// TIA Portal project "TruongKhuongDuy_20151451_DoanPLC_V17" (V17)
// Vorlageprojekt für das Buch mit Zielsystem S7-1200

(* hardware
DEVICE "S7-1200-Station_1"  S7-1200 Station
   slot 0: "Baugruppenträger_0"  Rack  V1.0
   slot 1: "PLC_1"  CPU 1211C DC/DC/DC  6ES7 211-1AE40-0XB0  V4.1
*)

// ===== PLC "PLC_1"  CPU 1211C DC/DC/DC =====

VAR_GLOBAL   // PLC tag table "Standard-Variablentabelle"
   "At exit" AT %I0.0 : Bool;
   "Start" AT %I0.1 : Bool;
   "Reset" AT %I0.2 : Bool;
   "Stop" AT %I0.3 : Bool;
   "Auto" AT %M20.0 : Bool;
   "Sensor 1" AT %I0.6 : Bool;
   "Sensor 4" AT %I0.7 : Bool;
   "Sensor 2" AT %I1.0 : Bool;
   "Sensor 3" AT %I1.1 : Bool;
   "Sensor box" AT %I1.2 : Bool;
   "Clamped" AT %I1.3 : Bool;
   "Limit" AT %I1.4 : Bool;
   "Detected 1" AT %I1.5 : Bool;
   "Moving Z1" AT %I1.6 : Bool;
   "Moving X1" AT %I1.7 : Bool;
   "Clamped 2" AT %I2.0 : Bool;
   "Limit 2" AT %I2.1 : Bool;
   "Detected 2" AT %I2.2 : Bool;
   "Moving Z2" AT %I2.3 : Bool;
   "Moving X2" AT %I2.4 : Bool;
   "Out Vision sensor" AT %ID30 : DInt;
   "Entry Converyor" AT %Q0.0 : Bool;
   "Alam siren" AT %Q0.1 : Bool;
   "Exit converyor" AT %Q0.2 : Bool;
   "Sotter 1 turn" AT %Q0.3 : Bool;
   "Sotter 1 belt" AT %Q0.4 : Bool;
   "Sotter 2 turn" AT %Q0.5 : Bool;
   "Sotter 2 belt" AT %Q0.6 : Bool;
   "Sotter 3 turn" AT %Q0.7 : Bool;
   "Sotter 3 belt" AT %Q1.0 : Bool;
   "Start light" AT %Q1.1 : Bool;
   "Reset light" AT %Q1.2 : Bool;
   "Stop light" AT %Q1.3 : Bool;
   "Belt Conveyor 1" AT %Q1.4 : Bool;
   "Belt Conveyor 2" AT %Q1.5 : Bool;
   "Box Conveyor" AT %Q1.6 : Bool;
   "Clamp 1" AT %Q1.7 : Bool;
   "Raise 1" AT %Q2.0 : Bool;
   "Mover Z1" AT %Q2.1 : Bool;
   "Mover X1" AT %Q2.2 : Bool;
   "Grab 1" AT %Q2.3 : Bool;
   "Clamp 2" AT %Q2.4 : Bool;
   "Raise 2" AT %Q2.5 : Bool;
   "Mover Z2" AT %Q2.6 : Bool;
   "Mover X2" AT %Q2.7 : Bool;
   "Grab 2" AT %Q3.0 : Bool;
   "Start Light ( Green)" AT %Q3.1 : Bool;
   "Reset Light ( Yellow)" AT %Q3.2 : Bool;
   "Stop Light ( Red)" AT %Q3.3 : Bool;
   "Stop Blade 1" AT %Q3.4 : Bool;
   "Counter 1" AT %QD30 : DInt;
   "Counter 2" AT %QD34 : DInt;
   "Counter 3" AT %QD38 : DInt;
   "Counter 4" AT %QD42 : DInt;
   "TG1" AT %M0.0 : Bool;
   "TG4" AT %M0.1 : Bool;
   "TG3" AT %M1.1 : Bool;
   "TG STOP CG" AT %M0.2 : Bool;
   "TG5" AT %M0.5 : Bool;
   "TG6" AT %M0.3 : Bool;
   "Tag_3" AT %M100.0 : Bool;
   "Tag_1" AT %M100.1 : Bool;
   "CB sensor4" AT %M100.3 : Bool;
   "Tag_2" AT %M101.1 : Bool;
   "Tag_4" AT %M100.2 : Bool;
   "Tag_5" AT %M100.4 : Bool;
   "Tag_6" AT %M100.7 : Bool;
   "Tag_8" AT %M100.6 : Bool;
   "Tag_9" AT %M200.0 : Bool;
   "Tag_10" AT %M200.1 : Bool;
   "Tag_11" AT %M200.2 : Bool;
   "Tag_12" AT %M200.3 : Bool;
   "Tag_13" AT %M200.4 : Bool;
   "Tag_14" AT %M200.7 : Bool;
   "Tag_15" AT %M200.6 : Bool;
   "Tag_16" AT %QD46 : DWord;
   "Tag_17" AT %M100.5 : Bool;
   "M_Stop" AT %M150.1 : Bool;
   "M_Reset" AT %M150.2 : Bool;
   "M_Start" AT %M150.0 : Bool;
   "M_exit" AT %M150.3 : Bool;
   "M_sensor1" AT %M150.4 : Bool;
   "M_sensor2" AT %M150.5 : Bool;
   "M_sensor3" AT %M150.6 : Bool;
   "M_sensor4" AT %M150.7 : Bool;
   "M_sensorbox" AT %M151.0 : Bool;
   "M_Auto" AT %M151.1 : Bool;
   "Tag_18" AT %M151.2 : Bool;
   "Tag_7" AT %M210.0 : Bool;
   "Emergency stop" AT %I0.4 : Bool;
END_VAR

// folder: System blocks/Program resources

DATA_BLOCK "IEC_Timer_0_DB"   // DB1
{ S7_Optimized_Access := 'TRUE' }
AUTHOR : Simatic
FAMILY : IEC
NAME : IEC_TMR
VERSION : 1.0
// stored: InstanceOfName IEC_TIMER
"IEC_TIMER"
BEGIN
END_DATA_BLOCK

DATA_BLOCK "IEC_Timer_0_DB_1"   // DB2
{ S7_Optimized_Access := 'TRUE' }
AUTHOR : Simatic
FAMILY : IEC
NAME : IEC_TMR
VERSION : 1.0
// stored: InstanceOfName IEC_TIMER
"IEC_TIMER"
BEGIN
END_DATA_BLOCK

DATA_BLOCK "IEC_Timer_0_DB_2"   // DB3
{ S7_Optimized_Access := 'TRUE' }
AUTHOR : Simatic
FAMILY : IEC
NAME : IEC_TMR
VERSION : 1.0
// stored: InstanceOfName IEC_TIMER
"IEC_TIMER"
BEGIN
END_DATA_BLOCK

DATA_BLOCK "IEC_Counter_0_DB_12"   // DB4
{ S7_Optimized_Access := 'TRUE' }
AUTHOR : Simatic
FAMILY : IEC
NAME : CNTR
VERSION : 1.0
// stored: InstanceOfName IEC_COUNTER
"IEC_COUNTER"
BEGIN
END_DATA_BLOCK

DATA_BLOCK "IEC_Counter_0_DB_16"   // DB5
{ S7_Optimized_Access := 'TRUE' }
AUTHOR : Simatic
FAMILY : IEC
NAME : CNTR
VERSION : 1.0
// stored: InstanceOfName IEC_COUNTER
"IEC_COUNTER"
BEGIN
END_DATA_BLOCK

DATA_BLOCK "IEC_Counter_0_DB_4"   // DB6
{ S7_Optimized_Access := 'TRUE' }
AUTHOR : Simatic
FAMILY : IEC
NAME : CNTR
VERSION : 1.0
// stored: InstanceOfName IEC_COUNTER
"IEC_COUNTER"
BEGIN
END_DATA_BLOCK

DATA_BLOCK "IEC_Counter_0_DB_2"   // DB7
{ S7_Optimized_Access := 'TRUE' }
AUTHOR : Simatic
FAMILY : IEC
NAME : CNTR
VERSION : 1.0
// stored: InstanceOfName IEC_COUNTER
"IEC_COUNTER"
BEGIN
END_DATA_BLOCK

DATA_BLOCK "IEC_Counter_0_DB_3"   // DB8
{ S7_Optimized_Access := 'TRUE' }
AUTHOR : Simatic
FAMILY : IEC
NAME : CNTR
VERSION : 1.0
// stored: InstanceOfName IEC_COUNTER
"IEC_COUNTER"
BEGIN
END_DATA_BLOCK

DATA_BLOCK "IEC_Timer_0_DB_20"   // DB9
{ S7_Optimized_Access := 'TRUE' }
AUTHOR : Simatic
FAMILY : IEC
NAME : IEC_TMR
VERSION : 1.0
// stored: InstanceOfName IEC_TIMER
"IEC_TIMER"
BEGIN
END_DATA_BLOCK

DATA_BLOCK "IEC_Timer_0_DB_10"   // DB10
{ S7_Optimized_Access := 'TRUE' }
AUTHOR : Simatic
FAMILY : IEC
NAME : IEC_TMR
VERSION : 1.0
// stored: InstanceOfName IEC_TIMER
"IEC_TIMER"
BEGIN
END_DATA_BLOCK

DATA_BLOCK "IEC_Timer_0_DB_11"   // DB11
{ S7_Optimized_Access := 'TRUE' }
AUTHOR : Simatic
FAMILY : IEC
NAME : IEC_TMR
VERSION : 1.0
// stored: InstanceOfName IEC_TIMER
"IEC_TIMER"
BEGIN
END_DATA_BLOCK

DATA_BLOCK "IEC_Timer_0_DB_13"   // DB12
{ S7_Optimized_Access := 'TRUE' }
AUTHOR : Simatic
FAMILY : IEC
NAME : IEC_TMR
VERSION : 1.0
// stored: InstanceOfName IEC_TIMER
"IEC_TIMER"
BEGIN
END_DATA_BLOCK

// folder: (top level)

FUNCTION "Sorting sation" : Void   // FC2, LAD
{ S7_Optimized_Access := 'TRUE' }
VERSION : 0.1
   VAR_TEMP   // added for the SCL form of the ladder/FBD networks
      _w1 : Bool;
   END_VAR
BEGIN

REGION Network 1: KHOI DONG
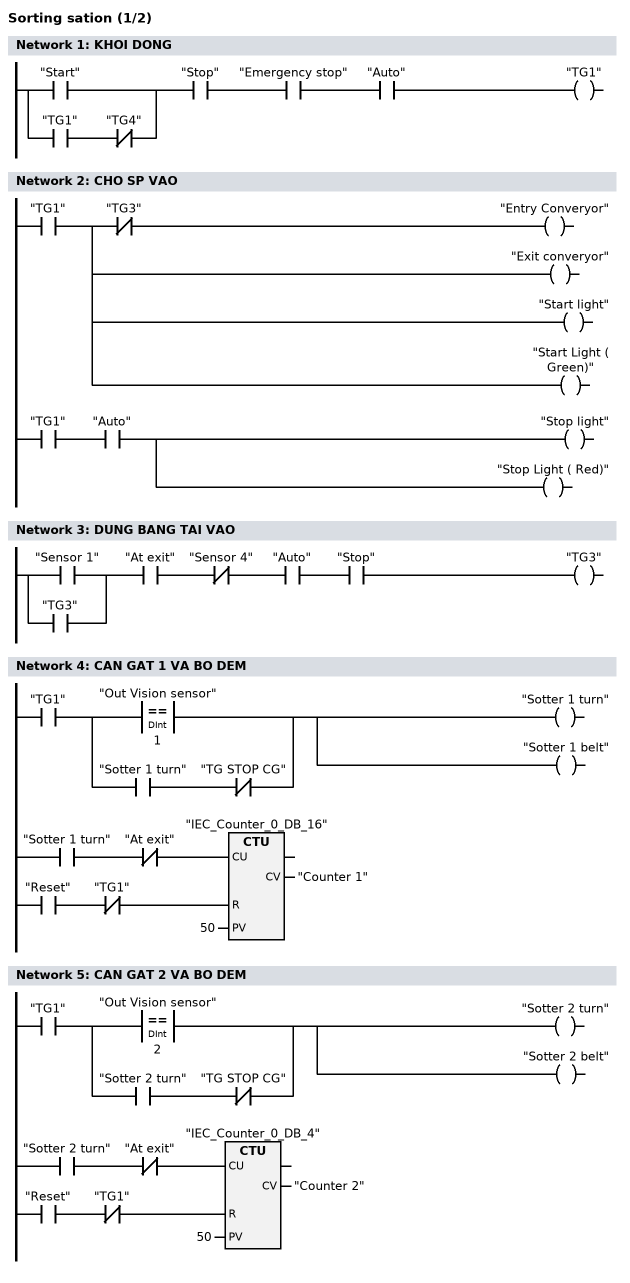
   RUNG wire#powerrail
      Contact( "Start" )
      wire#w1
      Contact( "Stop" )
      Contact( "Emergency stop" )
      Contact( "Auto" )
      Coil( "TG1" )
   END_RUNG
   RUNG wire#powerrail
      Contact( "TG1" )
      I_Contact( "TG4" )
   END_RUNG wire#w1
   // the same network as SCL:
   "TG1" := ("Start" OR ("TG1" AND NOT "TG4")) AND "Stop" AND "Emergency stop" AND "Auto";
END_REGION

REGION Network 2: CHO SP VAO
   RUNG wire#powerrail
      Contact( "TG1" )
      wire#w1
      I_Contact( "TG3" )
      Coil( "Entry Converyor" )
   END_RUNG
   RUNG wire#w1
      Coil( "Exit converyor" )
   END_RUNG
   RUNG wire#w1
      Coil( "Start light" )
   END_RUNG
   RUNG wire#w1
      Coil( "Start Light ( Green)" )
   END_RUNG
   RUNG wire#powerrail
      Contact( "TG1" )
      Contact( "Auto" )
      wire#w2
      Coil( "Stop light" )
   END_RUNG
   RUNG wire#w2
      Coil( "Stop Light ( Red)" )
   END_RUNG
   // the same network as SCL:
   "Entry Converyor" := "TG1" AND NOT "TG3";
   "Exit converyor" := "TG1";
   "Start light" := "TG1";
   "Start Light ( Green)" := "TG1";
   "Stop light" := "TG1" AND "Auto";
   "Stop Light ( Red)" := "Stop light";
END_REGION

REGION Network 3: DUNG BANG TAI VAO
   RUNG wire#powerrail
      Contact( "Sensor 1" )
      wire#w1
      Contact( "At exit" )
      I_Contact( "Sensor 4" )
      Contact( "Auto" )
      Contact( "Stop" )
      Coil( "TG3" )
   END_RUNG
   RUNG wire#powerrail
      Contact( "TG3" )
   END_RUNG wire#w1
   // the same network as SCL:
   "TG3" := ("Sensor 1" OR "TG3") AND "At exit" AND NOT "Sensor 4" AND "Auto" AND "Stop";
END_REGION

REGION Network 4: CAN GAT 1 VA BO DEM
   "Sotter 1 turn" := "TG1" AND (("Out Vision sensor" = 1) OR ("Sotter 1 turn" AND NOT "TG STOP CG"));
   "Sotter 1 belt" := "Sotter 1 turn";
   "IEC_Counter_0_DB_16".CTU(CU := "Sotter 1 turn" AND NOT "At exit",
                           R := "Reset" AND NOT "TG1",
                           PV := 50,
                           CV => "Counter 1");
END_REGION

REGION Network 5: CAN GAT 2 VA BO DEM
   "Sotter 2 turn" := "TG1" AND (("Out Vision sensor" = 2) OR ("Sotter 2 turn" AND NOT "TG STOP CG"));
   "Sotter 2 belt" := "Sotter 2 turn";
   "IEC_Counter_0_DB_4".CTU(CU := "Sotter 2 turn" AND NOT "At exit",
                           R := "Reset" AND NOT "TG1",
                           PV := 50,
                           CV => "Counter 2");
END_REGION

REGION Network 6: CAN GAT 3 VA BO DEM
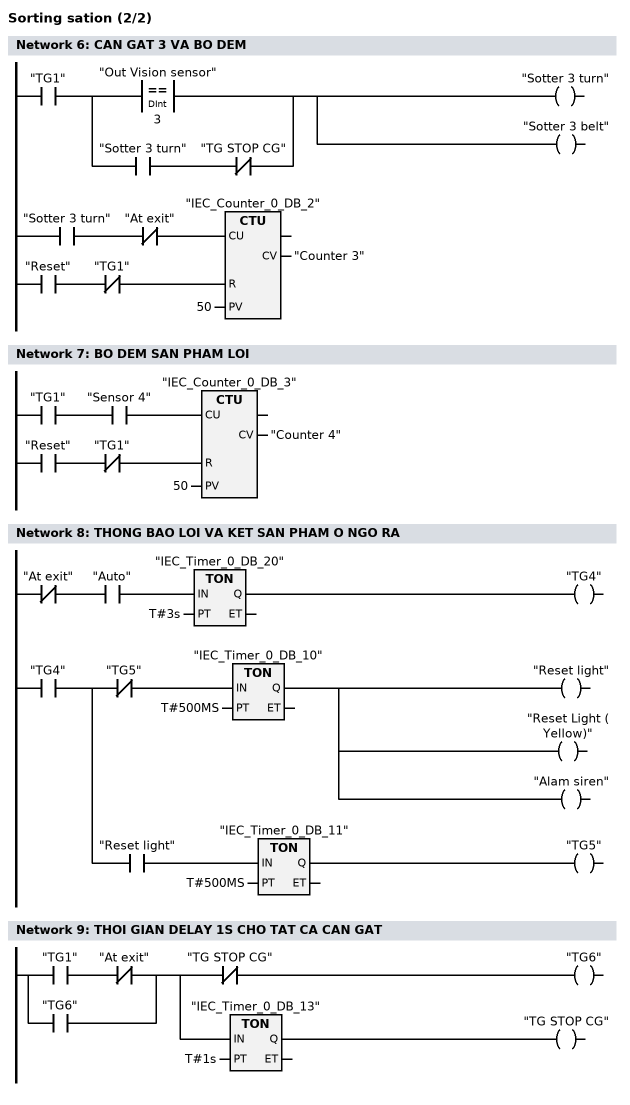
   "Sotter 3 turn" := "TG1" AND (("Out Vision sensor" = 3) OR ("Sotter 3 turn" AND NOT "TG STOP CG"));
   "Sotter 3 belt" := "Sotter 3 turn";
   "IEC_Counter_0_DB_2".CTU(CU := "Sotter 3 turn" AND NOT "At exit",
                           R := "Reset" AND NOT "TG1",
                           PV := 50,
                           CV => "Counter 3");
END_REGION

REGION Network 7: BO DEM SAN PHAM LOI
   "IEC_Counter_0_DB_3".CTU(CU := "TG1" AND "Sensor 4", R := "Reset" AND NOT "TG1", PV := 50, CV => "Counter 4");
END_REGION

REGION Network 8: THONG BAO LOI VA KET SAN PHAM O NGO RA
   "IEC_Timer_0_DB_20".TON(IN := NOT "At exit" AND "Auto", PT := T#3s);
   "TG4" := "IEC_Timer_0_DB_20".Q;
   "IEC_Timer_0_DB_10".TON(IN := "TG4" AND NOT "TG5", PT := T#500MS);
   "Reset light" := "IEC_Timer_0_DB_10".Q;
   "Reset Light ( Yellow)" := "IEC_Timer_0_DB_10".Q;
   "Alam siren" := "IEC_Timer_0_DB_10".Q;
   "IEC_Timer_0_DB_11".TON(IN := "TG4" AND "Reset light", PT := T#500MS);
   "TG5" := "IEC_Timer_0_DB_11".Q;
END_REGION

REGION Network 9: THOI GIAN DELAY 1S CHO TAT CA CAN GAT
   #_w1 := ("TG1" AND NOT "At exit") OR "TG6";
   "TG6" := #_w1 AND NOT "TG STOP CG";
   "IEC_Timer_0_DB_13".TON(IN := #_w1, PT := T#1s);
   "TG STOP CG" := "IEC_Timer_0_DB_13".Q;
END_REGION
END_FUNCTION

FUNCTION "Pick & Place 1" : Void   // FC3, LAD
{ S7_Optimized_Access := 'TRUE' }
VERSION : 0.1
   VAR_TEMP   // added for the SCL form of the ladder/FBD networks
      _w1 : Bool;
      _w2 : Bool;
      _w3 : Bool;
      _w4 : Bool;
      _w5 : Bool;
      _w6 : Bool;
   END_VAR
BEGIN

REGION Network 1: CHUONG TRINH
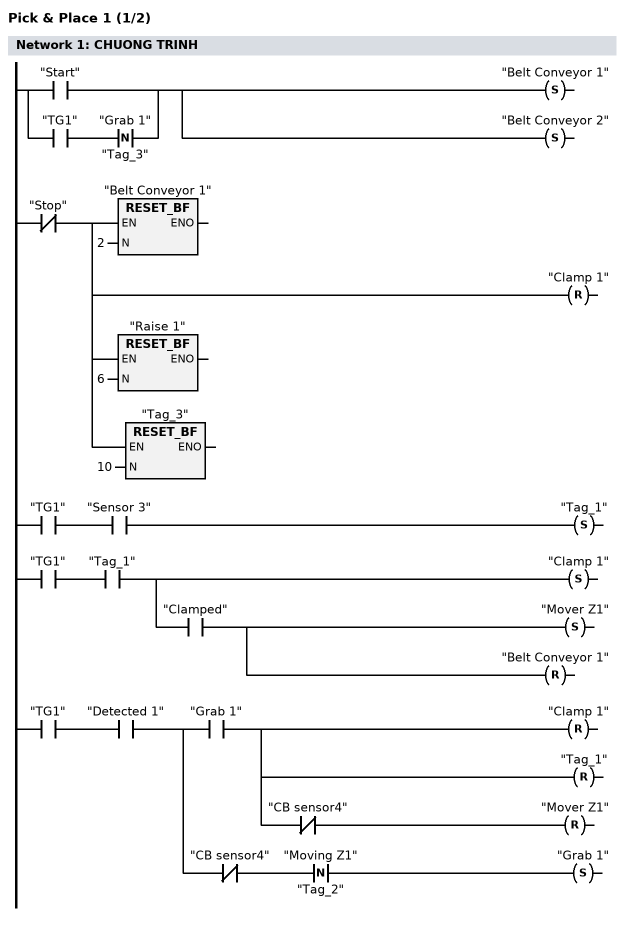
   // no SCL statement known for RBitfield: written as a call
   #_w1 := "TG1" AND NOT "Grab 1" AND "Tag_3";   // falling edge of "Grab 1"
   "Tag_3" := "Grab 1";
   IF "Start" OR #_w1 THEN
       "Belt Conveyor 1" := TRUE;
       "Belt Conveyor 2" := TRUE;
   END_IF;
   #_w2 := NOT "Stop";
   IF #_w2 THEN
       RESET_BF(operand := "Belt Conveyor 1", n := 2);
       "Clamp 1" := FALSE;
       RESET_BF(operand := "Raise 1", n := 6);
       RESET_BF(operand := "Tag_3", n := 10);
   END_IF;
   IF "TG1" AND "Sensor 3" THEN "Tag_1" := TRUE; END_IF;
   #_w3 := "TG1" AND "Tag_1";
   IF #_w3 THEN "Clamp 1" := TRUE; END_IF;
   IF #_w3 AND "Clamped" THEN
       "Mover Z1" := TRUE;
       "Belt Conveyor 1" := FALSE;
   END_IF;
   #_w4 := "TG1" AND "Detected 1";
   #_w5 := #_w4 AND "Grab 1";
   IF #_w5 THEN
       "Clamp 1" := FALSE;
       "Tag_1" := FALSE;
   END_IF;
   IF #_w5 AND NOT "CB sensor4" THEN "Mover Z1" := FALSE; END_IF;
   #_w6 := #_w4 AND NOT "CB sensor4" AND NOT "Moving Z1" AND "Tag_2";   // falling edge of "Moving Z1"
   "Tag_2" := "Moving Z1";
   IF #_w6 THEN "Grab 1" := TRUE; END_IF;
END_REGION

REGION Network 2
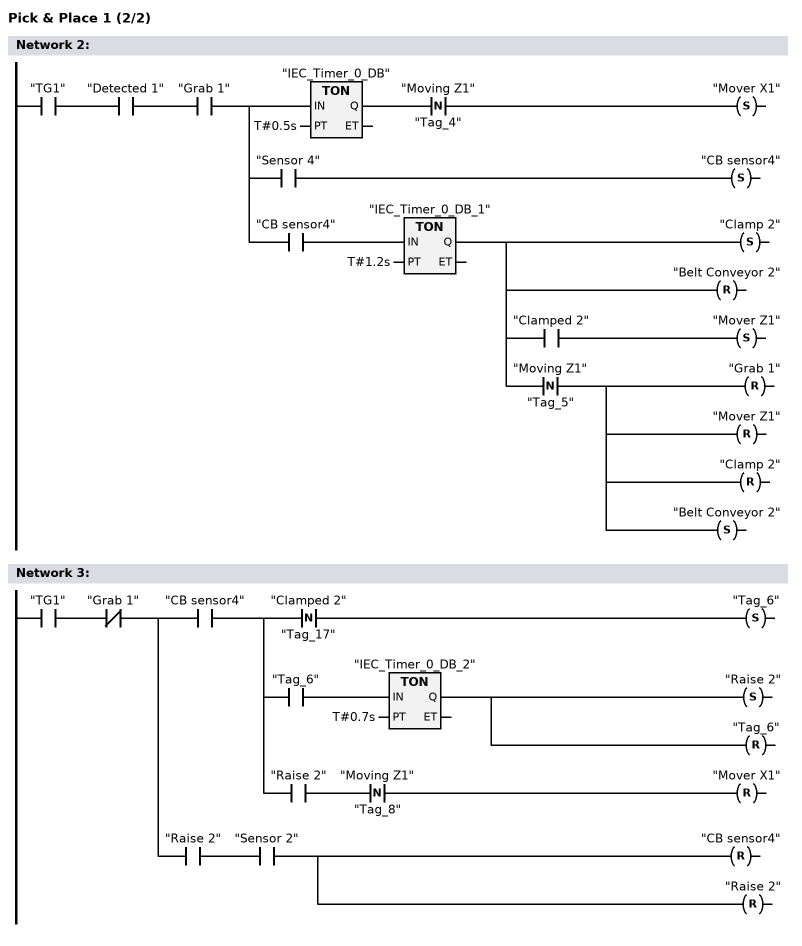
   #_w1 := "TG1" AND "Detected 1" AND "Grab 1";
   "IEC_Timer_0_DB".TON(IN := #_w1, PT := T#0.5s);
   #_w2 := "IEC_Timer_0_DB".Q AND NOT "Moving Z1" AND "Tag_4";   // falling edge of "Moving Z1"
   "Tag_4" := "Moving Z1";
   IF #_w2 THEN "Mover X1" := TRUE; END_IF;
   IF #_w1 AND "Sensor 4" THEN "CB sensor4" := TRUE; END_IF;
   "IEC_Timer_0_DB_1".TON(IN := #_w1 AND "CB sensor4", PT := T#1.2s);
   IF "IEC_Timer_0_DB_1".Q THEN
       "Clamp 2" := TRUE;
       "Belt Conveyor 2" := FALSE;
   END_IF;
   IF "IEC_Timer_0_DB_1".Q AND "Clamped 2" THEN "Mover Z1" := TRUE; END_IF;
   #_w3 := "IEC_Timer_0_DB_1".Q AND NOT "Moving Z1" AND "Tag_5";   // falling edge of "Moving Z1"
   "Tag_5" := "Moving Z1";
   IF #_w3 THEN
       "Grab 1" := FALSE;
       "Mover Z1" := FALSE;
       "Clamp 2" := FALSE;
       "Belt Conveyor 2" := TRUE;
   END_IF;
END_REGION

REGION Network 3
   #_w1 := "TG1" AND NOT "Grab 1";
   #_w2 := #_w1 AND "CB sensor4";
   #_w3 := #_w2 AND NOT "Clamped 2" AND "Tag_17";   // falling edge of "Clamped 2"
   "Tag_17" := "Clamped 2";
   IF #_w3 THEN "Tag_6" := TRUE; END_IF;
   "IEC_Timer_0_DB_2".TON(IN := #_w2 AND "Tag_6", PT := T#0.7s);
   IF "IEC_Timer_0_DB_2".Q THEN
       "Raise 2" := TRUE;
       "Tag_6" := FALSE;
   END_IF;
   #_w4 := #_w2 AND "Raise 2" AND NOT "Moving Z1" AND "Tag_8";   // falling edge of "Moving Z1"
   "Tag_8" := "Moving Z1";
   IF #_w4 THEN "Mover X1" := FALSE; END_IF;
   IF #_w1 AND "Raise 2" AND "Sensor 2" THEN
       "CB sensor4" := FALSE;
       "Raise 2" := FALSE;
   END_IF;
END_REGION
END_FUNCTION

FUNCTION "Pick & Place 2" : Void   // FC4, LAD
{ S7_Optimized_Access := 'TRUE' }
VERSION : 0.1
   VAR_TEMP   // added for the SCL form of the ladder/FBD networks
      _w1 : Bool;
      _w2 : Bool;
      _w3 : Bool;
      _w4 : Bool;
      _w5 : Bool;
      _w6 : Bool;
      _w7 : Bool;
      _w8 : Bool;
   END_VAR
BEGIN

REGION Network 1
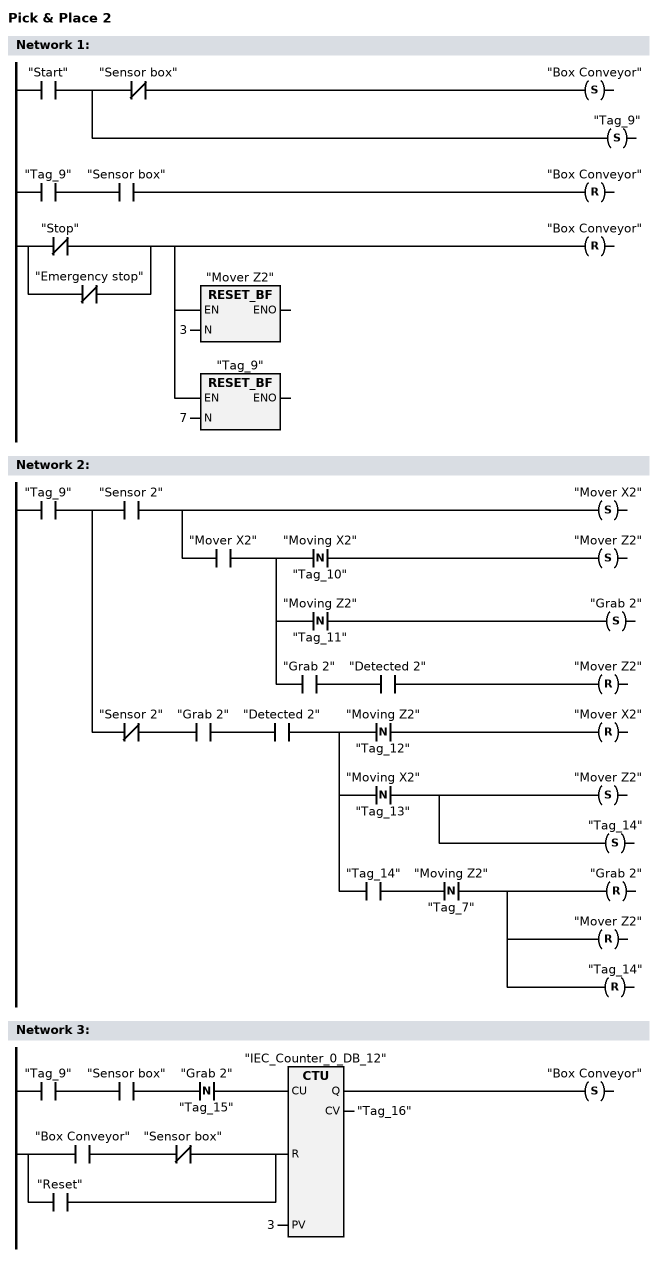
   // no SCL statement known for RBitfield: written as a call
   IF "Start" AND NOT "Sensor box" THEN "Box Conveyor" := TRUE; END_IF;
   IF "Start" THEN "Tag_9" := TRUE; END_IF;
   IF "Tag_9" AND "Sensor box" THEN "Box Conveyor" := FALSE; END_IF;
   IF NOT "Stop" OR NOT "Emergency stop" THEN "Box Conveyor" := FALSE; END_IF;
   #_w1 := NOT "Stop" OR NOT "Emergency stop";
   IF #_w1 THEN
       RESET_BF(operand := "Mover Z2", n := 3);
       RESET_BF(operand := "Tag_9", n := 7);
   END_IF;
END_REGION

REGION Network 2
   RUNG wire#powerrail
      Contact( "Tag_9" )
      wire#w1
      Contact( "Sensor 2" )
      wire#w2
      S_Coil( "Mover X2" )
   END_RUNG
   RUNG wire#w2
      Contact( "Mover X2" )
      wire#w3
      N_Contact(operand := "Moving X2", bit := "Tag_10")
      S_Coil( "Mover Z2" )
   END_RUNG
   RUNG wire#w3
      N_Contact(operand := "Moving Z2", bit := "Tag_11")
      S_Coil( "Grab 2" )
   END_RUNG
   RUNG wire#w3
      Contact( "Grab 2" )
      Contact( "Detected 2" )
      R_Coil( "Mover Z2" )
   END_RUNG
   RUNG wire#w1
      I_Contact( "Sensor 2" )
      Contact( "Grab 2" )
      Contact( "Detected 2" )
      wire#w4
      N_Contact(operand := "Moving Z2", bit := "Tag_12")
      R_Coil( "Mover X2" )
   END_RUNG
   RUNG wire#w4
      N_Contact(operand := "Moving X2", bit := "Tag_13")
      wire#w5
      S_Coil( "Mover Z2" )
   END_RUNG
   RUNG wire#w5
      S_Coil( "Tag_14" )
   END_RUNG
   RUNG wire#w4
      Contact( "Tag_14" )
      N_Contact(operand := "Moving Z2", bit := "Tag_7")
      wire#w6
      R_Coil( "Grab 2" )
   END_RUNG
   RUNG wire#w6
      R_Coil( "Mover Z2" )
   END_RUNG
   RUNG wire#w6
      R_Coil( "Tag_14" )
   END_RUNG
   // the same network as SCL:
   #_w1 := "Tag_9" AND "Sensor 2";
   IF #_w1 THEN "Mover X2" := TRUE; END_IF;
   #_w2 := #_w1 AND "Mover X2";
   #_w3 := #_w2 AND NOT "Moving X2" AND "Tag_10";   // falling edge of "Moving X2"
   "Tag_10" := "Moving X2";
   IF #_w3 THEN "Mover Z2" := TRUE; END_IF;
   #_w4 := #_w2 AND NOT "Moving Z2" AND "Tag_11";   // falling edge of "Moving Z2"
   "Tag_11" := "Moving Z2";
   IF #_w4 THEN "Grab 2" := TRUE; END_IF;
   IF #_w2 AND "Grab 2" AND "Detected 2" THEN "Mover Z2" := FALSE; END_IF;
   #_w5 := "Tag_9" AND NOT "Sensor 2" AND "Grab 2" AND "Detected 2";
   #_w6 := #_w5 AND NOT "Moving Z2" AND "Tag_12";   // falling edge of "Moving Z2"
   "Tag_12" := "Moving Z2";
   IF #_w6 THEN "Mover X2" := FALSE; END_IF;
   #_w7 := #_w5 AND NOT "Moving X2" AND "Tag_13";   // falling edge of "Moving X2"
   "Tag_13" := "Moving X2";
   IF #_w7 THEN
       "Mover Z2" := TRUE;
       "Tag_14" := TRUE;
   END_IF;
   #_w8 := #_w5 AND "Tag_14" AND NOT "Moving Z2" AND "Tag_7";   // falling edge of "Moving Z2"
   "Tag_7" := "Moving Z2";
   IF #_w8 THEN
       "Grab 2" := FALSE;
       "Mover Z2" := FALSE;
       "Tag_14" := FALSE;
   END_IF;
END_REGION

REGION Network 3
   #_w1 := "Tag_9" AND "Sensor box" AND NOT "Grab 2" AND "Tag_15";   // falling edge of "Grab 2"
   "Tag_15" := "Grab 2";
   "IEC_Counter_0_DB_12".CTU(CU := #_w1,
                           R := ("Box Conveyor" AND NOT "Sensor box") OR "Reset",
                           PV := 3,
                           CV => "Tag_16");
   IF "IEC_Counter_0_DB_12".Q THEN "Box Conveyor" := TRUE; END_IF;
END_REGION
END_FUNCTION

FUNCTION "MHJ-PLC-Lab-Function-S71200" : Void   // FC9000, SCL
{ S7_Optimized_Access := 'TRUE' }
VERSION : 0.1
   VAR_TEMP
      rdTimeReturn : Int;
      outputTime : DTL;
      SyncVal : Byte;
      forVal : Int;
      forVal_2 : Int;
      Value : Byte;
   END_VAR
   VAR CONSTANT
      CompVal : Byte := 16#34;
      Value_01 : Byte := 16#11;
      Value_01_DW : DWord := 16#A165_D992;
      Value_02_DW : DWord := 16#58BE_4401;
   END_VAR
BEGIN

   #Value:=PEEK(area := 16#82,
        dbNumber := 0,
        byteOffset := 511);
   #Value := #Value + 1;

   POKE(area := 16#82,
        dbNumber := 0,
        byteOffset := 511,
        value := #Value);

   POKE(area:=16#81,
        dbNumber:=0,
        byteOffset:=1016,
        value:=#Value_01_DW);
   POKE(area := 16#81,
        dbNumber := 0,
        byteOffset := 1020,
        value := #Value_02_DW);

   POKE(area := 16#81,
        dbNumber := 0,
        byteOffset := 511,
        value := B#16#00);

   FOR #forVal := 0 TO 120 DO
       FOR #forVal_2:=0 TO 10 DO
           #rdTimeReturn:=RD_SYS_T(#outputTime);
           #rdTimeReturn := WR_SYS_T(#outputTime);
           #rdTimeReturn := RD_SYS_T(#outputTime);
           #rdTimeReturn := WR_SYS_T(#outputTime);
       END_FOR;
       #SyncVal:= PEEK(area := 16#81,
                      dbNumber := 0,
                      byteOffset := 511);
       IF #SyncVal = #CompVal THEN
          GOTO M_1;
       END_IF;
   END_FOR;
   RETURN;

   M_1:
   POKE(area := 16#81,
        dbNumber := 0,
        byteOffset := 511,
        value := B#16#0);
END_FUNCTION

ORGANIZATION_BLOCK "Main"   // OB1, LAD, ProgramCycle
TITLE = "Main Program Sweep (Cycle)"
{ S7_Optimized_Access := 'TRUE' }
VERSION : 0.1
   VAR_INPUT
      Initial_Call : Bool;   // Initial call of this OB
      Remanence : Bool;   // =True, if remanent data are available
   END_VAR
   VAR_TEMP
      M_sensor2 : Bool;
   END_VAR
BEGIN

REGION Network 1: THU VIEN CONNECT
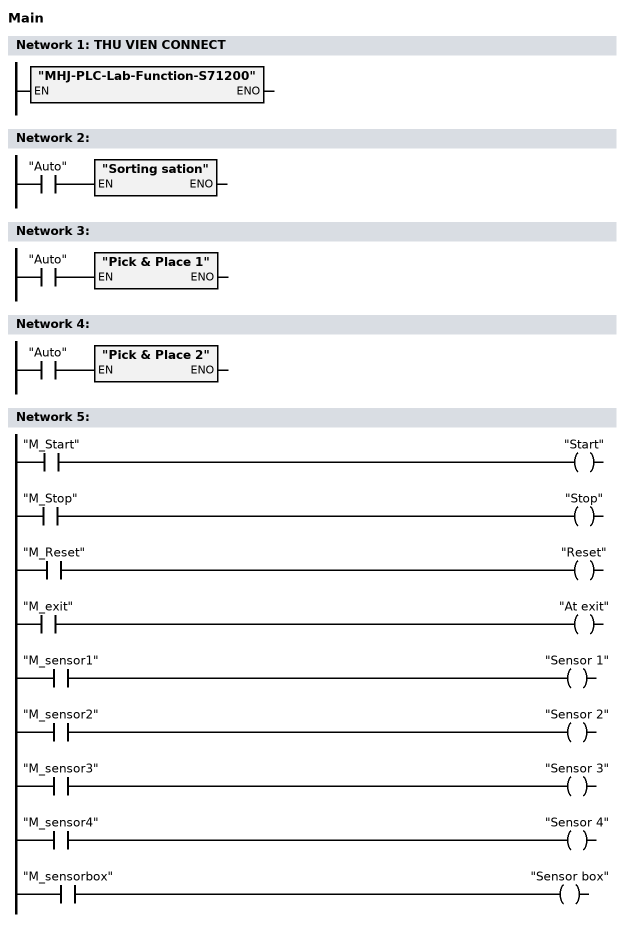
   RUNG wire#powerrail
      "MHJ-PLC-Lab-Function-S71200"()
   END_RUNG
   // the same network as SCL:
   "MHJ-PLC-Lab-Function-S71200"();
END_REGION

REGION Network 2
   RUNG wire#powerrail
      Contact( "Auto" )
      "Sorting sation"()
   END_RUNG
   // the same network as SCL:
   IF "Auto" THEN "Sorting sation"(); END_IF;
END_REGION

REGION Network 3
   RUNG wire#powerrail
      Contact( "Auto" )
      "Pick & Place 1"()
   END_RUNG
   // the same network as SCL:
   IF "Auto" THEN "Pick & Place 1"(); END_IF;
END_REGION

REGION Network 4
   RUNG wire#powerrail
      Contact( "Auto" )
      "Pick & Place 2"()
   END_RUNG
   // the same network as SCL:
   IF "Auto" THEN "Pick & Place 2"(); END_IF;
END_REGION

REGION Network 5
   RUNG wire#powerrail
      Contact( "M_Start" )
      Coil( "Start" )
   END_RUNG
   RUNG wire#powerrail
      Contact( "M_Stop" )
      Coil( "Stop" )
   END_RUNG
   RUNG wire#powerrail
      Contact( "M_Reset" )
      Coil( "Reset" )
   END_RUNG
   RUNG wire#powerrail
      Contact( "M_exit" )
      Coil( "At exit" )
   END_RUNG
   RUNG wire#powerrail
      Contact( "M_sensor1" )
      Coil( "Sensor 1" )
   END_RUNG
   RUNG wire#powerrail
      Contact( "M_sensor2" )
      Coil( "Sensor 2" )
   END_RUNG
   RUNG wire#powerrail
      Contact( "M_sensor3" )
      Coil( "Sensor 3" )
   END_RUNG
   RUNG wire#powerrail
      Contact( "M_sensor4" )
      Coil( "Sensor 4" )
   END_RUNG
   RUNG wire#powerrail
      Contact( "M_sensorbox" )
      Coil( "Sensor box" )
   END_RUNG
   // the same network as SCL:
   "Start" := "M_Start";
   "Stop" := "M_Stop";
   "Reset" := "M_Reset";
   "At exit" := "M_exit";
   "Sensor 1" := "M_sensor1";
   "Sensor 2" := "M_sensor2";
   "Sensor 3" := "M_sensor3";
   "Sensor 4" := "M_sensor4";
   "Sensor box" := "M_sensorbox";
END_REGION
END_ORGANIZATION_BLOCK